(* IEC 61131-3 sources: trust-platform/docs/upstream/probes, 9 files *)

(* ---- t07_type_var_same.st ---- *)
TYPE J1939 : STRUCT a : INT; END_STRUCT END_TYPE
VAR_GLOBAL
  J1939 : J1939;
END_VAR

(* ---- t10_func_noret.st ---- *)
FUNCTION F10 : INT
VAR_INPUT a : INT; END_VAR
END_FUNCTION

(* ---- t01_real_noexp.st ---- *)
FUNCTION_BLOCK T01
VAR r : REAL; END_VAR
r := 3E+38;
END_FUNCTION_BLOCK

(* ---- t04_empty_out.st ---- *)
FUNCTION_BLOCK FB4
VAR_INPUT a : INT; END_VAR
VAR_OUTPUT o : INT; q : BOOL; END_VAR
END_FUNCTION_BLOCK
FUNCTION_BLOCK T04
VAR x : FB4; END_VAR
x(a := 1, o =>, q =>);
END_FUNCTION_BLOCK

(* ---- t05_bit_lit.st ---- *)
FUNCTION_BLOCK T05
VAR dw : DWORD; b : BYTE; END_VAR
dw := dw AND 1;
IF dw = 0 THEN b := 1; END_IF
IF b <> 0 THEN b := b OR 16#80; END_IF
END_FUNCTION_BLOCK

(* ---- t06_prog.st ---- *)
PROGRAM P6
VAR_INPUT i : INT; END_VAR
VAR_OUTPUT o : INT; END_VAR
o := i;
END_PROGRAM
FUNCTION_BLOCK FB6
VAR_OUTPUT q : INT; END_VAR
END_FUNCTION_BLOCK
PROGRAM T06
VAR x : INT; f : FB6; END_VAR
P6(i := 1);
x := P6.o;
f(q => P6.i);
END_PROGRAM

(* ---- t08_ctu.st ---- *)
FUNCTION_BLOCK T08
VAR c : CTU; n : INT; END_VAR
c(CU := TRUE, RESET := FALSE, PV := n);
n := c.CV;
END_FUNCTION_BLOCK

(* ---- t09_implicit.st ---- *)
FUNCTION_BLOCK T09
VAR b : BYTE; i : INT; w : WORD; x : BOOL; r : REAL; a : ARRAY[0..3] OF INT; END_VAR
i := b;
w := i;
b := w;
x := 1;
i := a[b];
CASE b OF 0: i := 1; END_CASE
i := b * i;
END_FUNCTION_BLOCK

(* ---- t11_literal_assign.st ---- *)
FUNCTION_BLOCK T11
VAR b : BYTE := 255; w : WORD := 16#FFFF; END_VAR
b := 16#FF;   (* E203 cannot assign 'USINT' to 'BYTE', the initializer above is accepted *)
w := 16#FFFF; (* E203 cannot assign 'UINT' to 'WORD' *)
b := 255;     (* E203 cannot assign 'INT' to 'BYTE' *)
IF w = 16#FFFF THEN b := 0; END_IF (* E201 types are not comparable *)
END_FUNCTION_BLOCK
